{attribute 'qualified_only'}
{attribute 'strict'}
TYPE E_ScopeCommand : 
(
	eDefault := 0,
	ePause,
	eStop
) ;
END_TYPE

(* stored: DUT E_ScopeCommand: Id f7d57032-c135-4eaf-b917-804a27eda6f4 *)
